// TIA Portal V21 export
TYPE "Rcp_DataOut_Type"
   STRUCT
      Busy : Bool;
      Alarm_Active : Bool := FALSE;
      Warning_Timeout : Bool := FALSE;
      Warning_Active : Bool := FALSE;   // Notice to the operator
      Rcp_in_Work_Modified : Bool;   // Recipe in work modified but not saved in archive
      Rcp_ShowSaveReminder : Bool;   // Enable popup save reminder in the recipe pages
      Rcp_Changed : Bool;   // Changeover Done, recipe is changed
      PB_Enb_Load_in_Work : Bool;   // enable function in HMI
      PB_Enb_Load_in_Edit : Bool;   // enable function in HMI
      PB_Enb_Save_in_Archive : Bool;   // enable function in HMI
      PB_Enb_Save_in_Work : Bool;   // enable function in HMI
      PB_Enb_Copy : Bool;   // enable function in HMI
      Rcp_Saved_in_work_mem : Bool;
      Rcp_Saved_in_archive_mem : Bool;
      Rcp_last_recipe_edited : Int;
      Rcp_last_recipe_saved_in_work : Int;
      Rcp_show_popup_unsaved_recipe : Bool;
      Rcp_show_unsaved_recipe_PBloadFromWork : Bool;
      Rcp_show_unsaved_recipe_PBloadFromEdit : Bool;
      HMI_in_rcp_page : Bool;
      RCP_GEN_List { S7_SetPoint := 'True'} : Array[0.."K_NumMacchinaARicetta"] of "Rcp_Name_Type";
      RCP_rcp_edit_name { S7_SetPoint := 'True'} : String[30];   // used for KTP comfort
      RCP_rcp_dest_name { S7_SetPoint := 'True'} : String[30];   // used for KTP comfort
      RCP_Max : Int;
   END_STRUCT;
END_TYPE
